// TIA Portal V17 export
// export: Created 2024-09-15T12:30:31.8963496Z, ExportSetting WithDefaults, DisplayName Totally Integrated Automation Portal, DisplayVersion V17, DisplayName TIA Portal Openness, DisplayVersion V17, DisplayName TIA Portal Version Control Interface, DisplayVersion V17, DisplayName STEP 7 Professional, DisplayVersion V17, DisplayName STEP 7 Safety, DisplayVersion V17, DisplayName WinCC Professional, DisplayVersion V17
TYPE "typ_Alert_Message"
// stored: IsFailsafeCompliant false
   STRUCT
      ldt_ts : LDT;
      s_id : String;
      s_data : String;
      i_code : Int;
   END_STRUCT;
END_TYPE
